{attribute addProperty BoxType "EL5021-0000-0016"}
{attribute addProperty Id "Enable_latch_CBIT10.1251Set_counterBIT10.1253"}
{attribute addProperty CRC "1576471057"}
{attribute addProperty SizeInBites "16"}
{attribute addProperty SizeInBytes "2"}
TYPE Control_5DF70A11 :
STRUCT
	{attribute addProperty Name "Enable_latch_C"}
	Enable_latch_C : BIT;
	{attribute 'hide'}
	reserve_1 : BIT;
	{attribute addProperty Name "Set_counter"}
	Set_counter : BIT;
	{attribute 'hide'}
	reserve_2_BIT_0 : BIT;
	{attribute 'hide'}
	reserve_2_BIT_1 : BIT;
	{attribute 'hide'}
	reserve_2_BIT_2 : BIT;
	{attribute 'hide'}
	reserve_2_BIT_3 : BIT;
	{attribute 'hide'}
	reserve_2_BIT_4 : BIT;
	{attribute 'hide'}
	reserve_2_BIT_5 : BIT;
	{attribute 'hide'}
	reserve_2_BIT_6 : BIT;
	{attribute 'hide'}
	reserve_2_BIT_7 : BIT;
	{attribute 'hide'}
	reserve_2_BIT_8 : BIT;
	{attribute 'hide'}
	reserve_2_BIT_9 : BIT;
	{attribute 'hide'}
	reserve_2_BIT_10 : BIT;
	{attribute 'hide'}
	reserve_2_BIT_11 : BIT;
	{attribute 'hide'}
	reserve_2_BIT_12 : BIT;
END_STRUCT
END_TYPE

(* stored: Version 1.2.0.0, ProductVersion 3.1.4024.9
   DUT Control_5DF70A11: Id {50d1f658-c947-4abe-a801-40104fcc4e63} *)
